FUNCTION ROUND (* this function rounds a real down to n digits behind the comma. *)
  (* Standard: 61499-1 *)
  (* Version 1.0, 2026-09-17, Franz Höpfinger, Portiert aus OSCAT_basic ROUND.TcPOU (Franz: 'portiere diese Funktionen hier her') - setup.DECADES[LIMIT(0,N,8)] (globales Array, in diesem Projekt nicht vorhanden) durch direkte Berechnung via EXPT(10.0, N) ersetzt. Damit entfaellt auch die urspruengliche Begrenzung von N auf 0-8 (die nur wegen der Array-Grenzen noetig war). *)
  PACKAGE OSCAT::Basic::POUs::Mathematical;
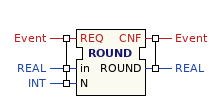
  EVENT_INPUT
    REQ WITH in, N;
  END_EVENT
  EVENT_OUTPUT
    CNF WITH ROUND;
  END_EVENT
  VAR_INPUT
    in : REAL;
    N : INT;
  END_VAR
  VAR_OUTPUT
    ROUND : REAL;
  END_VAR
  BODY IN ST:
PACKAGE OSCAT::Basic::POUs::Mathematical;

(* this function rounds a real down to n digits behind the comma. *)
FUNCTION ROUND : REAL
VAR_INPUT
	in : REAL;
	N : INT;
END_VAR
VAR
	X : REAL;
END_VAR

(*
 * version 1.5	25. oct. 2008 programmer 	hugo tested by	tobias
 * *
 * this function rounds a real down to n digits behind the comma.
 * Portiert 2026-09-17: setup.DECADES[LIMIT(0,N,8)] (Array in diesem Projekt nicht vorhanden) durch
 * direkte Berechnung via EXPT ersetzt - keine Begrenzung von N mehr auf 0-8.
 *)
X := EXPT(10.0, N);
ROUND := DINT_TO_REAL(REAL_TO_DINT(in * X)) / X;

END_FUNCTION

(* revision history hm	1. sep 2006	rev 1.0 original version
 * *
 * hm	2. dec 2007	rev 1.1 changed code for better performance
 * *
 * hm	8. jan 2008	rev 1.2 further improvement in performance
 * *
 * hm 11. mar. 2008	rev 1.3 corrected an error with negative numbers, use real_to_dint instead of trunc
 * *
 * hm	16. mar 2008	rev 1.4 added type conversion to avoid warning under codesys 3.0
 * *
 * hm	25. oct. 2008	rev 1.5 new code using global constants decades (hier ersetzt durch EXPT, siehe oben) *)
  END_BODY
END_FUNCTION
